Universal Robots PolyScope program: rq_is_motion_complete.urp

ProgramRoot directory=/home/rd/ursim-1.8/programs/Canevas; kinematics=(a=[0, -0.425, -0.39225, 0, 0, 0], d=[0.08916, 0, 0, 0.10915, 0.09465, 0.0823], alpha=[1.5708, 0, 0, 1.5708, -1.5708, 0], deltaTheta=[0, 0, 0, 0, 0, 0], status=notInitialized); name=rq_is_motion_complete; robotEnvironmentFileName=default
  MainProgram cartesianAcceleration=1.2; cartesianSpeed=0.25; jointAcceleration=1.3962634015954636; jointSpeed=1.0471975511965976; moveAsFastAsPossible=true; sharedProcessMoveBlendRadius=0.025; featureReference=(installationNameReference=Base); motionType=JOINT_SPACE
    Script type=0; expressionBranchNode=rq_is_motion_complete()
